FUNCTION "FC_ActionApDosage" : Void
{ S7_Optimized_Access := 'TRUE' }
VERSION : 0.1
   VAR_INPUT
      Surv_Benne : "S_DOSBENNE";
   END_VAR


BEGIN
END_FUNCTION

